TYPE EtcSlaveBase_82538BE2 :
STRUCT
END_STRUCT
END_TYPE

(* stored: Version 1.2.0.0, ProductVersion 3.1.4024.11
   DUT EtcSlaveBase_82538BE2: Id {5e854de9-2daa-4cc2-a8f0-acfbbee7fe4e} *)
